{attribute 'qualified_only'}
VAR_GLOBAL
	Flap_enable		AT%Q*:	BOOL;

	Flap_open		AT%Q*:	BOOL;

	Slit_enable		AT%Q*:	BOOL;

	slit_open		AT%Q*:	BOOL;
	
	OpenFlap		AT%I*: BOOL;
	CloseFlap		AT%I*: BOOL;
	OpenSlit		AT%I*: BOOL;
	CloseSlit		AT%I*: BOOL;

	ControlWord		AT%MW0: WORD;

END_VAR

(* stored: Version 1.1.0.1, ProductVersion 3.1.4024.0
   GVL GVL_Dome: Id {86115280-b596-42d6-92cd-0d7bfc111d95} *)
